// TIA Portal V16 export
// export: Created 2021-04-12T11:37:30.1360927Z, ExportSetting WithDefaults, DisplayName Totally Integrated Automation Portal, DisplayVersion V16 Update 1, DisplayName TIA Portal Version Control Interface, DisplayVersion V16, DisplayName TIA Portal Openness, DisplayVersion V16 Update 1, DisplayName SINAMICS Startdrive Advanced, DisplayVersion V16 Update 1, DisplayName SINAMICS Startdrive G130, G150, S120, S150, SINAMICS MV, S210, DisplayVersion V16 Update 1, DisplayName SINAMICS Startdrive G110M, G120, G120C, G120D, G120P, DisplayVersion V16 Update 1, DisplayName STEP 7 Professional, DisplayVersion V16 Update 1, DisplayName SIMATIC Energy Suite, DisplayVersion V16 Update 1, DisplayName STEP 7 Safety, DisplayVersion V16, DisplayName Simocode ES, DisplayVersion V16, DisplayName WinCC UA Professional, DisplayVersion V16 Update 1, DisplayName SIMATIC Visualization Architect, DisplayVersion V16
FUNCTION "AnalogOutputScaling" : Void   // FC1, LAD
{ S7_Optimized_Access := 'TRUE' }
VERSION : 0.1
// stored: AutoNumber true, IsIECCheckEnabled false, SetENOAutomatically false, UDAEnableTagReadback false
   VAR_INPUT
      rawValue : Int;   // Raw value of the analog input
      minSensor : Real;   // Minimum value of the sensor
      maxSensor : Real;   // Maximum value of the sensor
   END_VAR
   VAR_OUTPUT
      scaledValue : Real;   // Scaled value
   END_VAR
   VAR_TEMP
      temp_normalizedValue : Real;   // rawValue normalized to 0 - 100%
   END_VAR
   VAR CONSTANT
      MIN_ANALOG : Int := 0;
      MAX_ANALOG : Int := 27648;
   END_VAR
BEGIN

REGION Network 1
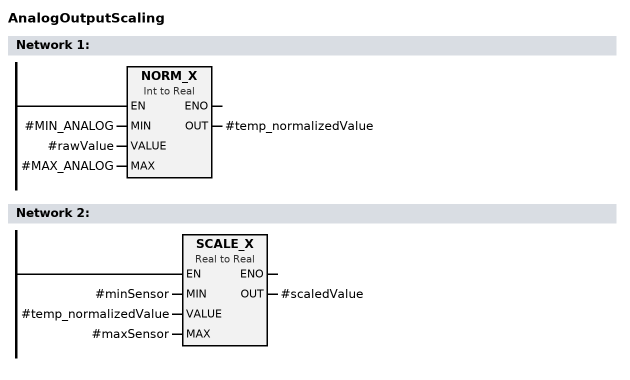
   RUNG wire#powerrail
      { S7_Templates := "[SrcType := Int, DestType := Real]" } Normalize(min := #MIN_ANALOG, value := #rawValue, max := #MAX_ANALOG, out => #temp_normalizedValue)
   END_RUNG
   // the same network as SCL:
   #temp_normalizedValue := NORM_X(MIN := #MIN_ANALOG, VALUE := #rawValue, MAX := #MAX_ANALOG);
END_REGION

REGION Network 2
   RUNG wire#powerrail
      { S7_Templates := "[SrcType := Real, DestType := Real]" } Scale(min := #minSensor, value := #temp_normalizedValue, max := #maxSensor, out => #scaledValue)
   END_RUNG
   // the same network as SCL:
   #scaledValue := SCALE_X(MIN := #minSensor, VALUE := #temp_normalizedValue, MAX := #maxSensor);
END_REGION
END_FUNCTION
